TYPE ST_Bottle :
STRUCT
	nId  : DINT ;
	fCurrentLevel : REAL;
	fTargetLevel : REAL;
	eLiquidType : E_LiquidType;
END_STRUCT
END_TYPE

(* stored: Version 1.1.0.1, ProductVersion 3.1.4024.16
   DUT ST_Bottle: Id {51fa5ce7-a434-4a11-839b-a5ea31d1b9b2} *)
